(* CoDeSys 2.3 export: ACTUATOR_CTRL.EXP *)

(* POU lib/ACTUATOR_CTRL, FBD *)
FUNCTION_BLOCK ACTUATOR_CTRL
VAR_INPUT
	xEMERGENCY					:	BOOL;
	iSTATE								:	INT;
	tSTATE4_DELAY_FOR_JUMP	:	TIME;
END_VAR
VAR_OUTPUT
	_xROTARY_MOTOR		:	BOOL;
	_xPUNCH					:	BOOL;
	_xLOWER_DRILL			:	BOOL;
	_xRAISE_DRILL			:	BOOL;
	_xDRILL					:	BOOL;
	_xDRILL_PUNCH			:	BOOL;
END_VAR
VAR
	ton_state4Delay		:	TON;
	rot1					:	BOOL;
	rot3					:	BOOL;
	rot7					:	BOOL;
	drill4					:	BOOL;
	drill5					:	BOOL;
END_VAR
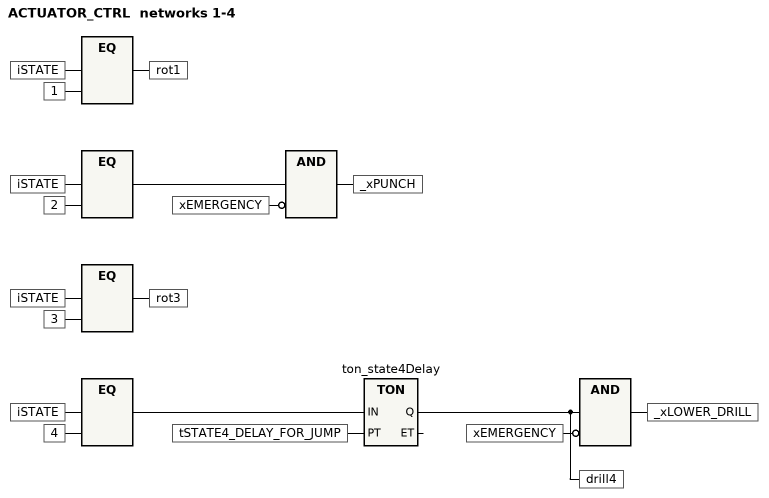
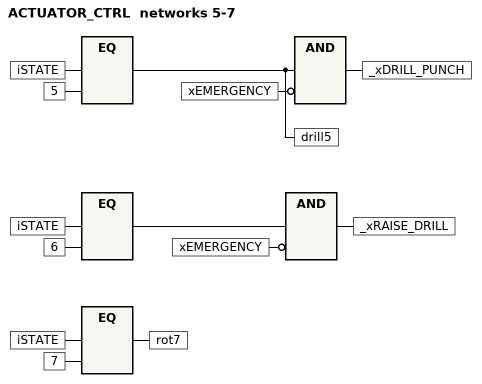
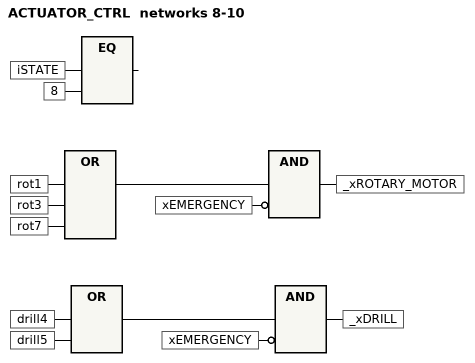
_FBD_ (* Function Block Diagram *)
NETWORK 1
	EQ(iSTATE, 1) => rot1
NETWORK 2
	AND(EQ(iSTATE, 2), NOT xEMERGENCY) => _xPUNCH
NETWORK 3
	EQ(iSTATE, 3) => rot3
NETWORK 4
	AND(<ton_state4Delay:TON(IN: EQ(iSTATE, 4), PT: tSTATE4_DELAY_FOR_JUMP) => drill4>, NOT xEMERGENCY) => _xLOWER_DRILL
NETWORK 5
	AND(<EQ(iSTATE, 5) => drill5>, NOT xEMERGENCY) => _xDRILL_PUNCH
NETWORK 6
	AND(EQ(iSTATE, 6), NOT xEMERGENCY) => _xRAISE_DRILL
NETWORK 7
	EQ(iSTATE, 7) => rot7
NETWORK 8
	EQ(iSTATE, 8)
NETWORK 9 rotaryCtrl: (* Because rotary is active in multiple states and can only be assigned once. *)
	AND(OR(rot1, rot3, rot7), NOT xEMERGENCY) => _xROTARY_MOTOR
NETWORK 10 drillCtrl: (* Because rotary is active in multiple states and can only be assigned once. *)
	AND(OR(drill4, drill5), NOT xEMERGENCY) => _xDRILL
_END_FBD_
(* the same logic as Structured Text *)
(* Network 1 *)
rot1 := iSTATE = 1;
(* Network 2 *)
_xPUNCH := (iSTATE = 2) AND NOT xEMERGENCY;
(* Network 3 *)
rot3 := iSTATE = 3;
(* Network 4 *)
ton_state4Delay(IN := iSTATE = 4, PT := tSTATE4_DELAY_FOR_JUMP);
drill4 := ton_state4Delay.Q;
_xLOWER_DRILL := ton_state4Delay.Q AND NOT xEMERGENCY;
(* Network 5 *)
drill5 := iSTATE = 5;
_xDRILL_PUNCH := drill5 AND NOT xEMERGENCY;
(* Network 6 *)
_xRAISE_DRILL := (iSTATE = 6) AND NOT xEMERGENCY;
(* Network 7 *)
rot7 := iSTATE = 7;
(* Network 8: see the listing above *)
(* Network 9 *)
_xROTARY_MOTOR := (rot1 OR rot3 OR rot7) AND NOT xEMERGENCY;
(* Network 10 *)
_xDRILL := (drill4 OR drill5) AND NOT xEMERGENCY;
END_FUNCTION_BLOCK
